ABB RAPID module: mfc_test_path1.mod

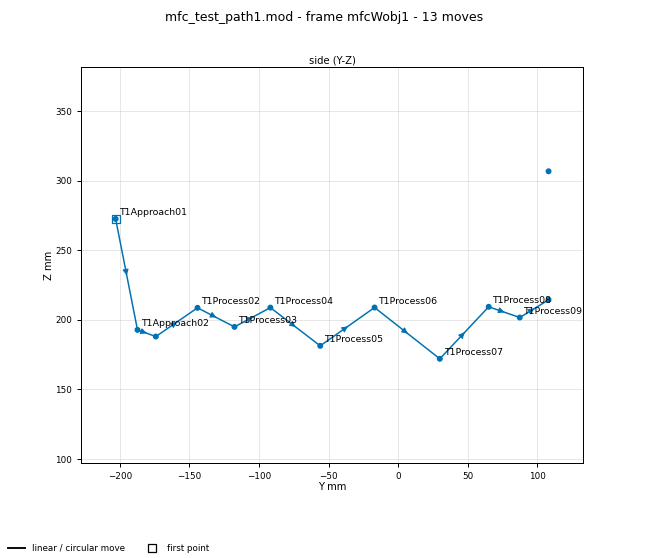
[picture p0: tool path of mfc_test_path1.mod in frame mfcWobj1, 13 of 14 moves have a stored position in this frame; points joined in program order, loops and branches not executed]
%%%
  VERSION: 1
  LANGUAGE: ENGLISH
%%%

MODULE mfc_test_path1

!This module is generated by RobotWare Machining FC V3.000. DO NOT EDIT.
!Any changes to this module will be lost when the RW Machining FC application is re-run and the program is exported.
LOCAL VAR robtarget T1Approach01 := [[508.71,-202.98,272.5],[0.000464213,0.796213,-0.605016,-0.000736645],[-1,-1,-2,0],[9E+09,9E+09,9E+09,9E+09,9E+09,9E+09]];
LOCAL VAR robtarget T1Approach02 := [[514.41,-187.29,192.81],[0.00046518,0.796217,-0.60501,-0.000738573],[-1,-1,-2,0],[9E+09,9E+09,9E+09,9E+09,9E+09,9E+09]];
LOCAL VAR robtarget T1Approach03 := [[514.41,-174.1,188.01],[0.000460651,0.796225,-0.604999,-0.000729966],[-1,-1,-2,0],[9E+09,9E+09,9E+09,9E+09,9E+09,9E+09]];
LOCAL VAR robtarget T1Process01  := [[514.4,-172.64,188],[0.000446613,0.796226,-0.604998,-0.000685263],[-1,-1,-2,0],[9E+09,9E+09,9E+09,9E+09,9E+09,9E+09]];
LOCAL VAR robtarget T1Process02  := [[514.34,-144.18,208.65],[0.000519177,0.796244,-0.604975,-0.000864234],[-1,-1,-2,0],[9E+09,9E+09,9E+09,9E+09,9E+09,9E+09]];
LOCAL VAR robtarget T1Process03  := [[514.35,-117.6,194.95],[0.000479273,0.796246,-0.604972,-0.00077805],[-1,-1,-2,0],[9E+09,9E+09,9E+09,9E+09,9E+09,9E+09]];
LOCAL VAR robtarget T1Process04  := [[514.34,-91.83,208.8],[0.000447091,0.796245,-0.604974,-0.000724376],[-1,-1,-2,0],[9E+09,9E+09,9E+09,9E+09,9E+09,9E+09]];
LOCAL VAR robtarget T1Process05  := [[514.37,-56.02,181.34],[0.000365649,0.796241,-0.604979,-0.000587182],[-1,-1,-2,0],[9E+09,9E+09,9E+09,9E+09,9E+09,9E+09]];
LOCAL VAR robtarget T1Process06  := [[514.34,-16.99,208.86],[0.000364398,0.796244,-0.604975,-0.000583088],[-1,0,-2,0],[9E+09,9E+09,9E+09,9E+09,9E+09,9E+09]];
LOCAL VAR robtarget T1Process07  := [[514.34,29.86,172.02],[0.000378565,0.796233,-0.60499,-0.000598426],[0,0,-2,0],[9E+09,9E+09,9E+09,9E+09,9E+09,9E+09]];
LOCAL VAR robtarget T1Process08  := [[514.32,64.98,209.38],[0.000414984,0.796231,-0.604992,-0.000631874],[0,0,-2,0],[9E+09,9E+09,9E+09,9E+09,9E+09,9E+09]];
LOCAL VAR robtarget T1Process09  := [[514.3,87.28,201.68],[0.000445599,0.796242,-0.604978,-0.000656885],[0,0,-2,0],[9E+09,9E+09,9E+09,9E+09,9E+09,9E+09]];
LOCAL VAR robtarget T1Process10  := [[514.3,107.98,214.36],[0.000423327,0.796238,-0.604983,-0.000635365],[0,0,-2,0],[9E+09,9E+09,9E+09,9E+09,9E+09,9E+09]];
LOCAL VAR robtarget T1Withdraw01 := [[514.29,107.97,244.2],[0.000424694,0.796241,-0.604979,-0.000637076],[0,0,-2,0],[9E+09,9E+09,9E+09,9E+09,9E+09,9E+09]];
LOCAL VAR robtarget T1Withdraw02 := [[514.27,107.97,306.71],[0.000485436,0.796243,-0.604977,-0.000691136],[0,0,-2,0],[9E+09,9E+09,9E+09,9E+09,9E+09,9E+09]];
LOCAL VAR num n1ForceX := 0;
LOCAL VAR num n1ForceY := 0;
LOCAL VAR num n1ForceZ := -10;


PROC run_test_path1 (bool bRecover, bool bSpindleOn)
	FCDeact;

	IF bRecover = true THEN
		FCCalib  mfcTool1_LD \Recovery;
	ELSE
		FCCalib  mfcTool1_LD;
	ENDIF

	IF bSpindleOn = true THEN
		SpindleOn;
	ENDIF

	MoveL T1Approach01, v50, z1,mfcTool1\wobj :=mfcWobj1;
	MoveL T1Approach02, v50, z1,mfcTool1\wobj :=mfcWobj1;
	MoveL T1Approach03, v50, fine,mfcTool1\wobj :=mfcWobj1;

	FCPress1LStart T1Process01, v50 \Fx:= n1ForceX \Fy:= n1ForceY \Fz:= n1ForceZ,50 \ForceFrameRef:=FC_REFFRAME_TOOL \ForceChange:=50 \DampingTune:=100 \TimeOut:=5, \UseSpdFFW, \PosSupvDist:=9e9, z1, mfcTool1 \wobj:=mfcWobj1;
	FCPressL T1Process02, v50, 10, z1, mfcTool1, \wobj:=mfcWobj1;
	FCPressL T1Process03, v50, 10, z1, mfcTool1, \wobj:=mfcWobj1;
	FCPressL T1Process04, v50, 10, z1, mfcTool1, \wobj:=mfcWobj1;
	FCPressL T1Process05, v50, 10, z1, mfcTool1, \wobj:=mfcWobj1;
	FCPressL T1Process06, v50, 10, z1, mfcTool1, \wobj:=mfcWobj1;
	FCPressL T1Process07, v50, 10, z1, mfcTool1, \wobj:=mfcWobj1;
	FCPressL T1Process08, v50, 10, z1, mfcTool1, \wobj:=mfcWobj1;
	FCPressL T1Process09, v50, 10, z1, mfcTool1, \wobj:=mfcWobj1;
	FCPressL T1Process10, v50, 10, z1, mfcTool1, \wobj:=mfcWobj1;

	FCPressLEnd T1Withdraw01,v50,\ForceChange :=50,\ZeroContactValue := 5;
	MoveL T1Withdraw02, v50, z1,mfcTool1\wobj :=mfcWobj1;

	IF bSpindleOn = true THEN
		SpindleOff;
	ENDIF

ENDPROC

ENDMODULE
